// Mitsubishi GX Works2 project: FINAL2.0   PLC: FX3G

// global labels: Global1
VAR_GLOBAL
  Switch7 AT X007 : BOOL;
  LIGHT1 AT Y001 : BOOL;
  Switch5 AT X005 : BOOL;
  LIGHT0 AT Y000 : BOOL;
  Honey AT D1200 : REAL;
  Oat AT D1300 : REAL;
  Protein AT D1400 : REAL;
  Switch3 AT X003 : BOOL;
END_VAR
VAR_GLOBAL CONSTANT
  YouAre5 : REAL := 5.0;
END_VAR
VAR_GLOBAL
  ClasicBar AT M2 : BOOL;
  YouGaveHoney AT D2000 : REAL;
  YouGaveOat AT D2100 : REAL;
  YouGaveProtein AT D2200 : REAL;
  MoreThen5 AT M3 : BOOL;
END_VAR
VAR_GLOBAL CONSTANT
  YouAre10 : REAL := 10.0;
END_VAR
VAR_GLOBAL
  ProteinBar AT M4 : BOOL;
  OutputAnalogGood AT M6 : BOOL;
END_VAR
VAR_GLOBAL CONSTANT
  GreaterThen400 : REAL := 400.0;
END_VAR
VAR_GLOBAL
  EnoughOatClasic AT M7 : BOOL;
END_VAR
VAR_GLOBAL CONSTANT
  GreaterThen120 : REAL := 400;
END_VAR
VAR_GLOBAL
  EnoughHoneyClasic AT M8 : BOOL;
  EnoughproteinClasic AT M9 : BOOL;
END_VAR
VAR_GLOBAL CONSTANT
  GreaterThen160 : REAL := 160;
END_VAR
VAR_GLOBAL
  EnoughOatPro AT M10 : BOOL;
END_VAR
VAR_GLOBAL CONSTANT
  GreaterThen240 : REAL := 240.0;
END_VAR
VAR_GLOBAL
  EnoughHoneyPro AT M11 : BOOL;
END_VAR
VAR_GLOBAL CONSTANT
  GreaterThen320 : REAL := 320;
END_VAR
VAR_GLOBAL
  EnoughProteinPro AT M12 : BOOL;
  Light3 AT Y003 : BOOL;
  TimerMixing AT TC1 : BOOL;
  Sec5 AT K50 : INT;
  ToBake AT M13 : BOOL;
  StartBakingSwitch2 AT X002 : BOOL;
  ForBlink AT M14 : BOOL;
  BlinkTimerClasic AT M15 : BOOL;
  BlinkTimerProtein AT M16 : BOOL;
  Sec4 AT K40 : INT;
END_VAR
VAR_GLOBAL CONSTANT
  Seconds4 : REAL := 40;
  BackingClassicTime : REAL := 40;
END_VAR
VAR_GLOBAL
  FinishBacking AT M17 : BOOL;
  StartPacking AT M18 : BOOL;
  FirstSnack AT CC1 : BOOL;
  Light4 AT Y004 : BOOL;
END_VAR
VAR_GLOBAL CONSTANT
  YouAre7 : REAL := 7.0;
END_VAR
VAR_GLOBAL
  WeFinishPackingSnacks AT M40 : BOOL;
  TotalSnackPacks AT CC8 : BOOL;
END_VAR
VAR_GLOBAL CONSTANT
  Startwith0 : INT;
  BakingClassicTime : REAL := 40;
END_VAR
VAR_GLOBAL
  Flickering1 AT M50 : BOOL;
  Sec05 AT K5 : INT;
  NURA1 AT TC2 : BOOL;
  NURA2 AT TC3 : BOOL;
  LIGHT2 AT Y002 : BOOL;
  NURA3 AT TC6 : BOOL;
  TimerMixingTS AT TS1 : BOOL;
  NURA1TS AT TS2 : BOOL;
  NURA2TS AT TS3 : BOOL;
  Mixinglight AT M300 : BOOL;
END_VAR
VAR_GLOBAL CONSTANT
  test : REAL := 100000;
END_VAR
VAR_GLOBAL
  DgimaAnalog AT M22 : BOOL;
  bartype AT D8280 : INT;
  classicFlikcering AT TC4 : BOOL;
  ProteinFlickering AT TC5 : BOOL;
  Switch6 AT X006 : BOOL;
  classicflickeringTS AT TS4 : BOOL;
  proteinflickeringTS AT TS5 : BOOL;
  Flickering2 AT M60 : BOOL;
  NURA4 AT TC7 : BOOL;
  NURA3TS AT TS6 : BOOL;
  NURA4TS AT TS7 : BOOL;
  Switch0 AT X000 : BOOL;
END_VAR
VAR_GLOBAL CONSTANT
  Snack1 : INT := 1;
END_VAR
VAR_GLOBAL
  Count7Snacks AT CS2 : BOOL;
END_VAR
VAR_GLOBAL CONSTANT
  finishedSnacks : INT := 8;
END_VAR
VAR_GLOBAL
  FinishedAllSnacks AT M20 : BOOL;
  NumOfPackets AT CC3 : BOOL;
END_VAR
VAR_GLOBAL CONSTANT
  PackCounter : REAL := 1;
END_VAR
VAR_GLOBAL
  Light4Off AT M70 : BOOL;
  PackReady AT D2500 : REAL;
  biggestOat AT M200 : BOOL;
  biggestHoney AT M210 : BOOL;
  biggestProtein AT M220 : BOOL;
END_VAR
VAR_GLOBAL CONSTANT
  YouAre400 : REAL := 400;
END_VAR
VAR_GLOBAL
  AnalogOutput AT D8282 : INT;
  Bartypeholder2 AT D1600 : REAL;
  bartypeholder4 AT D3001 : INT;
  TypeHolder AT D4001 : INT;
  WeReset AT M100 : BOOL;
  Count8Snacks AT CC2 : BOOL;
  FinishedResetingAll AT M101 : BOOL;
  Count8Snacks1 AT CS2 : BOOL;
  TimerClassicBar AT TC1 : BOOL;
  WeReset1 AT M101 : BOOL;
  LIGHT11 AT Y006 : BOOL;
  LIGHT6 AT Y006 : BOOL;
  Second3timer AT TC8 : BOOL;
  Sec2 AT K2 : INT;
  TS8 : BOOL;
  Holderfor2sec AT TS8 : BOOL;
  resetMLow AT M290 : BOOL;
  Enought2produceclasic AT M285 : BOOL;
  Enought2producepro AT M286 : BOOL;
  gomix AT M301 : BOOL;
  HoneyBegin AT D7000 : REAL;
  OatBegin AT D7002 : REAL;
  proteinBegin AT D7004 : REAL;
  begin_analog_input AT M400 : BOOL;
  invalid_input AT M407 : BOOL;
END_VAR
VAR_GLOBAL CONSTANT
  HoneyBegin1 : REAL := 800;
  OatBegin1 : REAL := 800;
  proteinBegin1 : REAL := 800;
END_VAR
VAR_GLOBAL
  BlinkTime AT D1212 : INT;
  readytoblink AT M333 : BOOL;
  moveto2 AT D1510 : REAL;
END_VAR
VAR_GLOBAL CONSTANT
  PacksDecimal : REAL := 40;
END_VAR

// task Task_01 (event TRUE, interval 0, priority 31): POU_01

PROGRAM POU_01
(* structured ladder/FBD written out as ST: instructions are called as NAME(EN, inputs, outputs); _pN, _eN, _tN stand for wires *)
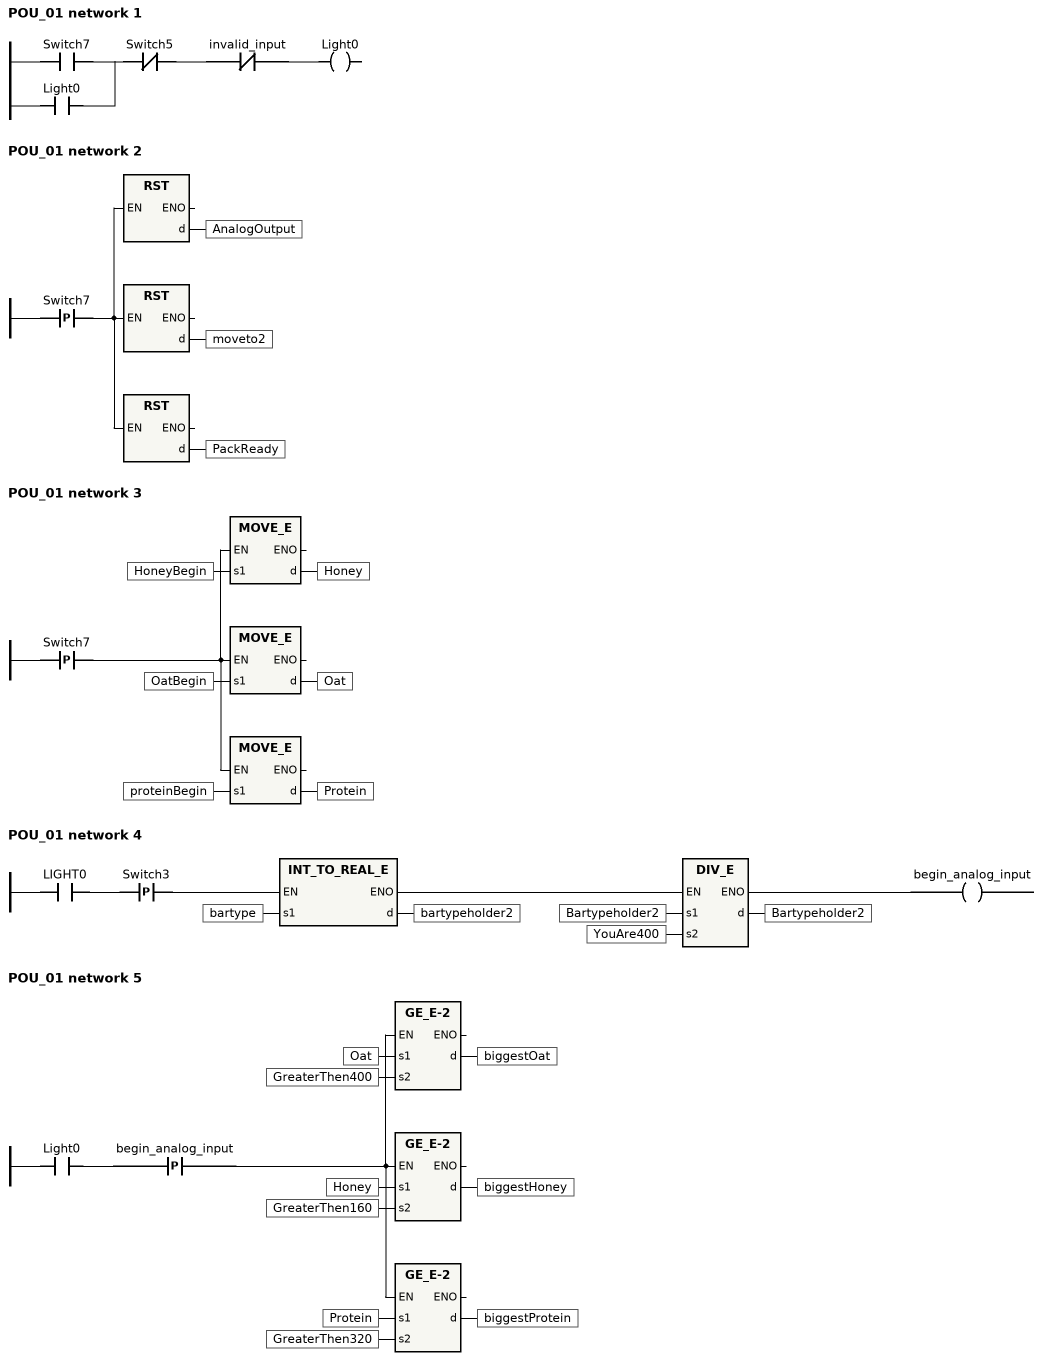
(* network 1 *)
Light0 := ((Switch7 OR Light0) AND NOT Switch5) AND NOT invalid_input;
(* network 2 *)
_p1 := LDP(TRUE, Switch7);
RST(_p1, AnalogOutput);
RST(_p1, moveto2);
RST(_p1, PackReady);
(* network 3 *)
_p1 := LDP(TRUE, Switch7);
MOVE_E(_p1, HoneyBegin, Honey);
MOVE_E(_p1, OatBegin, Oat);
MOVE_E(_p1, proteinBegin, Protein);
(* network 4 *)
_e1 := INT_TO_REAL_E(LIGHT0 AND LDP(TRUE, Switch3), bartype, bartypeholder2);
_e2 := DIV_E(_e1, Bartypeholder2, YouAre400, Bartypeholder2);
begin_analog_input := _e2;
(* network 5 *)
_p1 := Light0 AND LDP(TRUE, begin_analog_input);
GE_E(_p1, Oat, GreaterThen400, biggestOat);
GE_E(_p1, Honey, GreaterThen160, biggestHoney);
GE_E(_p1, Protein, GreaterThen320, biggestProtein);
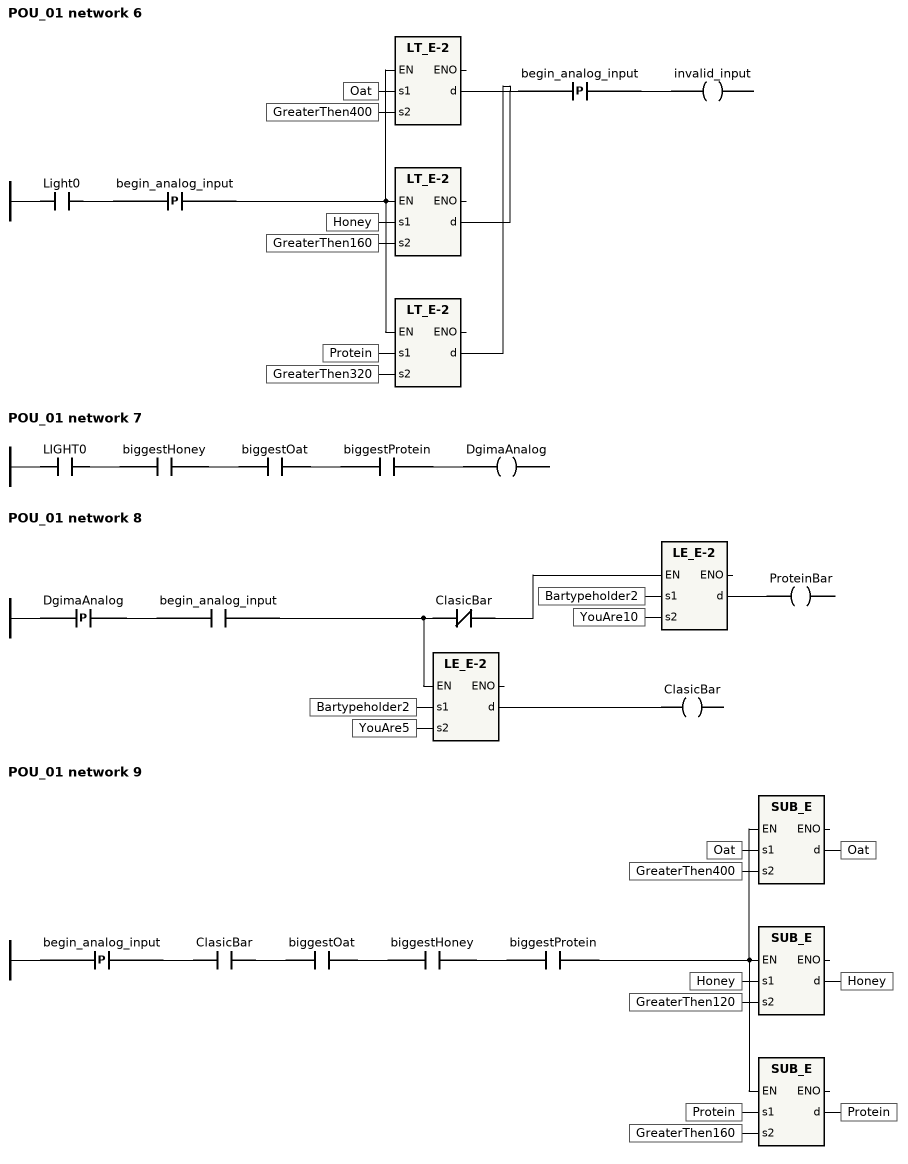
(* network 6 *)
_p1 := Light0 AND LDP(TRUE, begin_analog_input);
LT_E(_p1, Oat, GreaterThen400, _t2);
LT_E(_p1, Honey, GreaterThen160, _t3);
LT_E(_p1, Protein, GreaterThen320, _t4);
invalid_input := (_t2 OR _t3 OR _t4) AND LDP(TRUE, begin_analog_input);
(* network 7 *)
DgimaAnalog := LIGHT0 AND biggestHoney AND biggestOat AND biggestProtein;
(* network 8 *)
_p1 := LDP(TRUE, DgimaAnalog) AND begin_analog_input;
LE_E(_p1, Bartypeholder2, YouAre5, _t2);
ClasicBar := _t2;
LE_E(_p1 AND NOT ClasicBar, Bartypeholder2, YouAre10, _t3);
ProteinBar := _t3;
(* network 9 *)
_p1 := LDP(TRUE, begin_analog_input) AND ClasicBar AND biggestOat AND biggestHoney AND biggestProtein;
SUB_E(_p1, Oat, GreaterThen400, Oat);
SUB_E(_p1, Honey, GreaterThen120, Honey);
SUB_E(_p1, Protein, GreaterThen160, Protein);
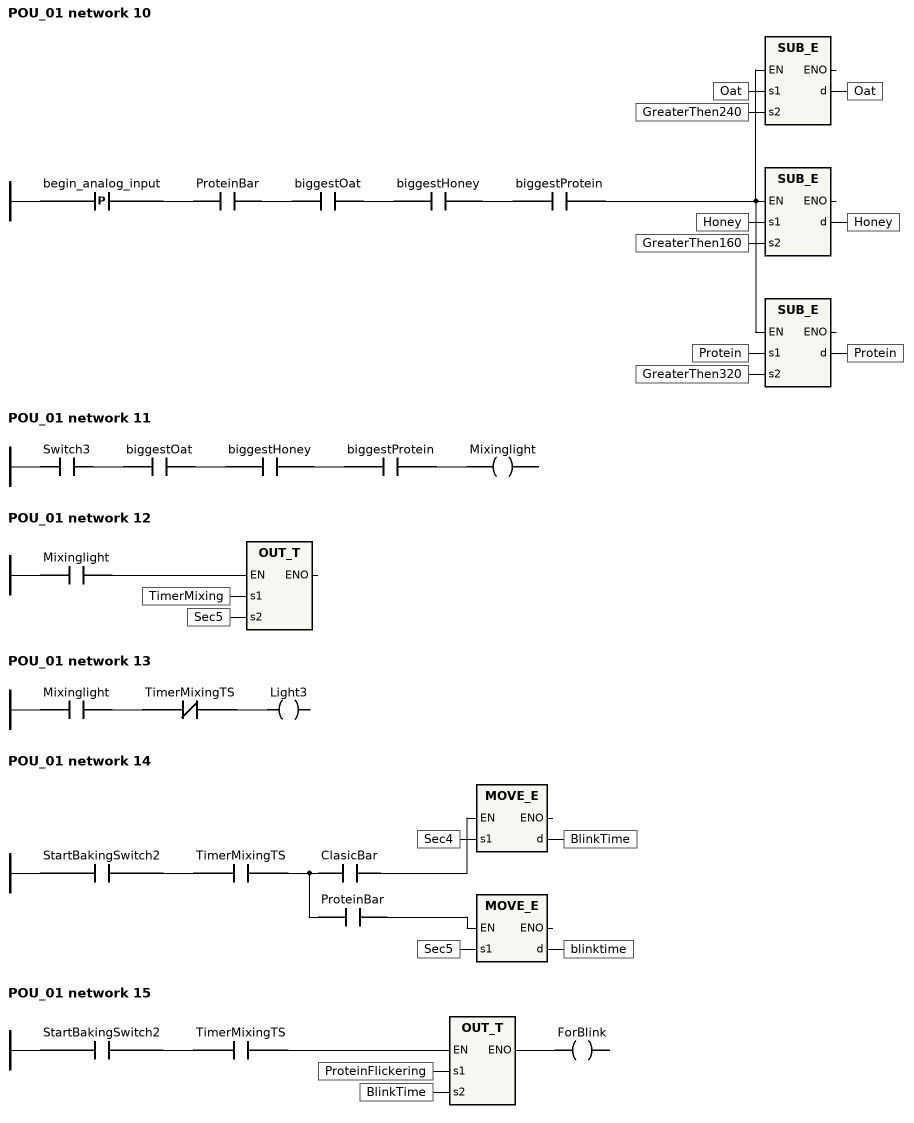
(* network 10 *)
_p1 := LDP(TRUE, begin_analog_input) AND ProteinBar AND biggestOat AND biggestHoney AND biggestProtein;
SUB_E(_p1, Oat, GreaterThen240, Oat);
SUB_E(_p1, Honey, GreaterThen160, Honey);
SUB_E(_p1, Protein, GreaterThen320, Protein);
(* network 11 *)
Mixinglight := Switch3 AND biggestOat AND biggestHoney AND biggestProtein;
(* network 12 *)
OUT_T(Mixinglight, TimerMixing, Sec5);
(* network 13 *)
Light3 := Mixinglight AND NOT TimerMixingTS;
(* network 14 *)
_p1 := StartBakingSwitch2 AND TimerMixingTS;
MOVE_E(_p1 AND ClasicBar, Sec4, BlinkTime);
MOVE_E(_p1 AND ProteinBar, Sec5, blinktime);
(* network 15 *)
_e1 := OUT_T(StartBakingSwitch2 AND TimerMixingTS, ProteinFlickering, BlinkTime);
ForBlink := _e1;
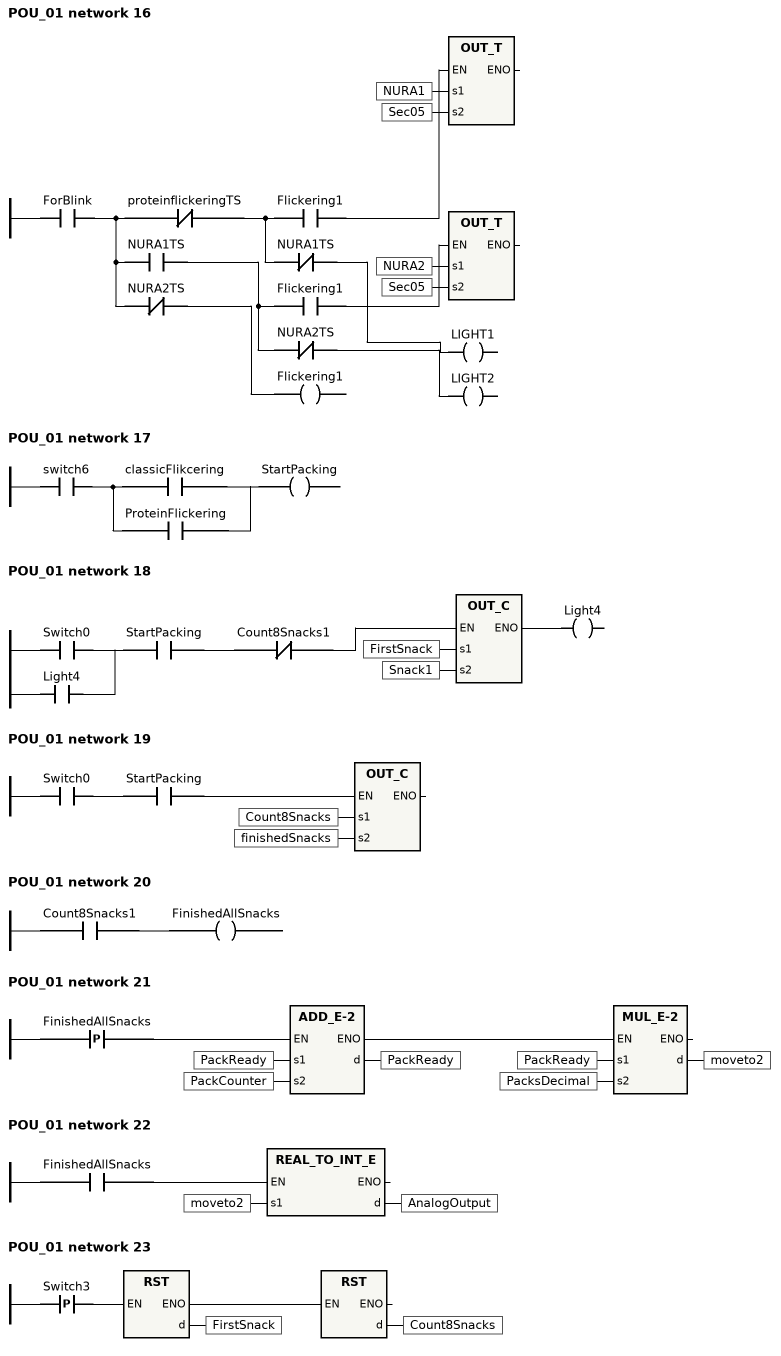
(* network 16 *)
_p1 := ForBlink AND NOT proteinflickeringTS;
OUT_T(_p1 AND Flickering1, NURA1, Sec05);
LIGHT1 := _p1 AND NOT NURA1TS;
_p2 := ForBlink AND NURA1TS;
OUT_T(_p2 AND Flickering1, NURA2, Sec05);
LIGHT2 := _p2 AND NOT NURA2TS;
Flickering1 := ForBlink AND NOT NURA2TS;
(* network 17 *)
StartPacking := (switch6 AND classicFlikcering) OR (switch6 AND ProteinFlickering);
(* network 18 *)
_e1 := OUT_C(((Switch0 OR Light4) AND StartPacking) AND NOT Count8Snacks1, FirstSnack, Snack1);
Light4 := _e1;
(* network 19 *)
OUT_C(Switch0 AND StartPacking, Count8Snacks, finishedSnacks);
(* network 20 *)
FinishedAllSnacks := Count8Snacks1;
(* network 21 *)
_e1 := ADD_E(LDP(TRUE, FinishedAllSnacks), PackReady, PackCounter, PackReady);
MUL_E(_e1, PackReady, PacksDecimal, moveto2);
(* network 22 *)
REAL_TO_INT_E(FinishedAllSnacks, moveto2, AnalogOutput);
(* network 23 *)
_e1 := RST(LDP(TRUE, Switch3), FirstSnack);
RST(_e1, Count8Snacks);
END_PROGRAM
